// TIA Portal V20 export
DATA_BLOCK "BK02"   // DB191
// stored: MemoryReserve 100
   VAR
      "X10-1 ELECTRODE FIX RIGHT TOP BACKWARD" : Bool;
      "X10-2 ELECTRODE FIX RIGHT TOP FORWARD" : Bool;
      "X12-1 ELECTRODE FIX RIGHT BTM BACKWARD" : Bool;
      "X12-2 ELECTRODE FIX RIGHT BTM FORWARD" : Bool;
      "X14-1 ELECTRODE FIX RIGHT TOP PRESSURE SWITCH" : Bool;
      "X14-2 ELECTRODE FIX RIGHT BTM PRESSURE SWITCH" : Bool;
      "X16-1 ELECTRODE CUTTER BACKWARD" : Bool;
      "X16-2 ELECTRODE CUTTER FORWARD" : Bool;
   END_VAR
BEGIN
END_DATA_BLOCK
